FUNCTION_BLOCK ConditionIF_ELSE (* Lua Test FB for IF statement *)
  (* Standard: 61499-2; Description: IF  is TRUE when a > b IF_ELSE is TRUE when b > c ELSE is TRUE when non of the above trigger Copyright (c) 2019 Jan Holzweber This program and the accompanying materials are made available under the terms of the Eclipse Public License 2.0 which is available at https://www.eclipse.org/legal/epl-2.0/ SPDX-License-Identifier: EPL-2.0 *)
  (* Version 1.0, 2019-06-05, jholz *)
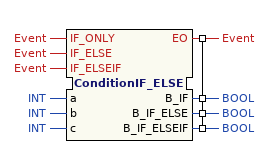
  EVENT_INPUT
    IF_ONLY;
    IF_ELSE;
    IF_ELSEIF;
  END_EVENT
  EVENT_OUTPUT
    EO WITH B_IF, B_IF_ELSE, B_IF_ELSEIF;
  END_EVENT
  VAR_INPUT
    a : INT;
    b : INT;
    c : INT;
  END_VAR
  VAR_OUTPUT
    B_IF : BOOL;
    B_IF_ELSE : BOOL;
    B_IF_ELSEIF : BOOL;
  END_VAR
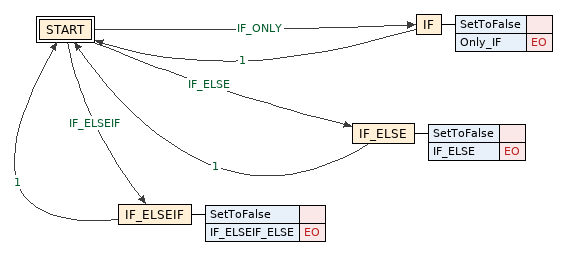
  EC_STATES
    START; (* Initial State *)
    IF : SetToFalse, Only_IF -> EO;
    IF_ELSE : SetToFalse, IF_ELSE -> EO;
    IF_ELSEIF : SetToFalse, IF_ELSEIF_ELSE -> EO;
  END_STATES
  EC_TRANSITIONS
    START TO IF := IF_ONLY;
    START TO IF_ELSE := IF_ELSE;
    START TO IF_ELSEIF := IF_ELSEIF;
    IF TO START := 1;
    IF_ELSE TO START := 1;
    IF_ELSEIF TO START := 1;
  END_TRANSITIONS
  ALGORITHM Only_IF IN ST: (* new algorithm *)
if a > b then
	B_IF := true;
end_if;
  END_ALGORITHM
  ALGORITHM IF_ELSE IN ST: (* new algorithm *)
if a > b then
	B_IF := true;
elsif b > c then
	B_IF_ELSEIF := true;
end_if;
  END_ALGORITHM
  ALGORITHM IF_ELSEIF_ELSE IN ST: (* new algorithm *)
if a > b then
	B_IF := true;
elsif b > c then
	B_IF_ELSEIF := true;
else
	B_IF_ELSE :=true;
end_if;
  END_ALGORITHM
  ALGORITHM SetToFalse IN ST: (* new algorithm *)
B_IF := false;
B_IF_ELSEIF := false;
B_IF_ELSE :=false;
  END_ALGORITHM
END_FUNCTION_BLOCK
